(* IEC 61131-3 sources: Industry-PLC-LLM/data/PLCBEAD_repo/PLCBEAD_PLCEmbed-main/PLC-BEAD/Source/GEB/SHL1, 1 file *)

(* ---- SHL1.ST ---- *)
FUNCTION SHL1:DWORD

	VAR_INPUT
		IN :	DWORD;
		N :	INT;
	END_VAR

	SHL1 := SHR(DWORD#16#FF_FF_FF_FF,32-N) OR SHL(IN,N);

END_FUNCTION

PROGRAM program0

	VAR
		IN :	DWORD;
		N :	INT;
		CEIL5_OUT : DWORD;
	END_VAR

  	CEIL5_OUT := SHL1(IN, N);

END_PROGRAM
